{attribute 'qualified_only'}
{attribute 'strict'}
TYPE E_Event :
(
	Alarm := 0,
	Message := 1,
	Warning := 2
);
END_TYPE

(* stored: Version 1.1.0.1, ProductVersion 3.1.4024.16
   DUT E_Event: Id {3eaee391-5b69-42ed-ba6e-529fd1469cc5} *)
